{attribute addProperty BoxType "KL3042"}
{attribute addProperty Id "Channel_1Channel_B0A8062F00Channel_2Channel_B0A8062F00"}
{attribute addProperty CRC "3175726068"}
{attribute addProperty SizeInBites "0"}
{attribute addProperty SizeInBytes "0"}
TYPE KL3042_BD49BBF4 :
STRUCT
	{attribute addProperty Name "Channel_1"}
	Channel_1 : Channel_B0A8062F;
	{attribute addProperty Name "Channel_2"}
	Channel_2 : Channel_B0A8062F;
END_STRUCT
END_TYPE

(* stored: Version 1.2.0.0, ProductVersion 3.1.4024.9
   DUT KL3042_BD49BBF4: Id {340728f1-6352-4923-adc7-1605bbd78c2d} *)
